// TIA Portal V20 export
DATA_BLOCK "PM2"   // DB274
// stored: MemoryReserve 100
   VAR
      "STACK #2 NG CLAMP MOVER CLOSE" : Bool;
      "STACK #2 NG CLAMP MOVER OPEN" : Bool;
      "STACK #2 NG CLAMP LEFT CLOSE" : Bool;
      "STACK #2 NG CLAMP LEFT OPEN" : Bool;
      "STACK #2 NG CLAMP RIGHT CLOSE" : Bool;
      "STACK #2 NG CLAMP RIGHT OPEN" : Bool;
      "STAKC #2 NG CLAMP Z-AXIS UP" : Bool;
      "STAKC #2 NG CLAMP Z-AXIS DOWN" : Bool;
      "STAKC #2 NG CLAMP MOVER FORWARD" : Bool;
      "STAKC #2 NG CLAMP MOVER BACKWARD" : Bool;
      "STACK #2 NG BOX LIFT UP" : Bool;
      "STACK #2 NG BOX LIFT DOWN" : Bool;
      "STACK #2 NG BOX LOCK UP" : Bool;
      "STACK #2 NG BOX LOCK DOWN" : Bool;
      "JR OUT P&P#2 CLAMP CLOSE" : Bool;
      "JR OUT P&P#2 CLAMP OPEN" : Bool;
   END_VAR
BEGIN
END_DATA_BLOCK
